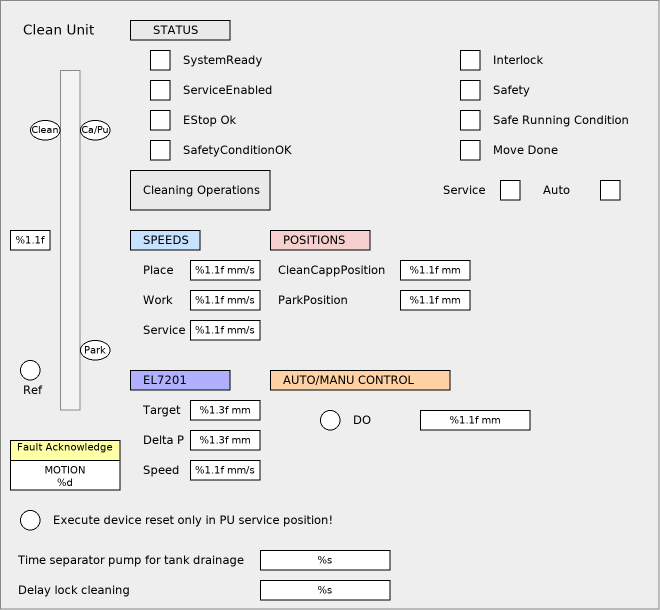
VISUALIZATION _VISU_CLEAN_CU  // 660x610
VAR_IN_OUT
  m_Inst : INT;               (*visu instance*) 
END_VAR
    Rectangle (0,0 660x610)
    Polyline (200,380)
    Rectangle (130,370 100x20)
    Rectangle (270,370 180x20)
    Rectangle (270,230 100x20)
    Rectangle (130,230 70x20)
    Rectangle (280,370 170x20), "AUTO/MANU CONTROL"
    Polyline (440,380)
    Ellipse (20,360 20x20), colour toggle: PRG_MACHINE.fb_CleaningCU[m_Inst].bL_ReferenceSensor
    Rectangle (20,380 30x20), "Ref"
    Scrollbar (60,70 20x340)
        p3598130195: -0.01
        p2245068023: 0.6
        p1057716461: PRG_MACHINE.fb_CleaningCU[m_Inst].fB_Axis.fO_ActualPosition
    Rectangle (10,230 40x20), "%1.1f", text variable: 1000 * PRG_MACHINE.fb_CleaningCU[m_Inst].fB_Axis.fO_ActualPosition
    Rectangle (140,230 70x20), "SPEEDS"
    Polyline (130,240)
    Polyline (340,240)
    Rectangle (280,230 90x20), "POSITIONS"
    Rectangle (190,400 70x20), "%1.3f mm", text variable: 1000 * PRG_MACHINE.fb_CleaningCU[m_Inst].fB_Axis.fI_TargetPosition
    Rectangle (140,400 70x20), "Target"
    Rectangle (140,460 70x20), "Speed"
    Rectangle (190,460 70x20), "%1.1f mm/s", text variable: 1000 * PRG_MACHINE.fb_CleaningCU[m_Inst].fB_Axis.fI_SpeedLimit
    Rectangle (140,370 90x20), "EL7201"
    Rectangle (140,430 70x20), "Delta P"
    Rectangle (190,430 70x20), "%1.3f mm", text variable: 1000 * PRG_MACHINE.fb_CleaningCU[m_Inst].fB_Axis.fL_Delta_P
    Ellipse (30,120 30x20), "Clean", colour toggle: PRG_MACHINE.fb_CleaningCU[m_Inst].pInPosCappingClean
    Ellipse (80,340 30x20), "Park", colour toggle: PRG_MACHINE.fb_CleaningCU[m_Inst].pInPosPark
    Ellipse (80,120 30x20), "Ca/Pu", colour toggle: PRG_MACHINE.fb_CleaningCU[m_Inst].pInPosCappingClean
    Rectangle (20,20 110x20), "Clean Unit"
    Rectangle (10,440 110x50), "Fault Acknowledge", colour toggle: (PRG_MACHINE.fb_CleaningCU[m_Inst].wL_ErrorCode) <> 0
    RoundedRectangle (10,460 110x30), "%d", text variable: PRG_MACHINE.fB_CleaningCU[m_Inst].wL_ErrorCode
        tap PRG_MACHINE.sADS_CleanAxis[iCPr_MAP_Cp_CuAxis[m_Inst]].bI_FaultAck
    RoundedRectangle (10,460 110x20), "MOTION"
    Rectangle (130,170 140x40)
    Rectangle (130,20 100x20)
    Polyline (130,30)
    Polyline (230,30)
    Rectangle (150,20 60x20), "STATUS"
    RoundedRectangle (150,80 20x20), colour toggle: PRG_MACHINE.fb_CleanProcess[m_Inst].bI_UsrService
    RoundedRectangle (150,110 20x20), colour toggle: PRG_MACHINE.bL_IO_EStopOK
    RoundedRectangle (150,140 20x20), colour toggle: PRG_MACHINE.fB_Machine.bI_SafetyOk
    RoundedRectangle (460,140 20x20), colour toggle: NOT PRG_MACHINE.fb_CleaningCU[m_Inst].bL_Busy
    RoundedRectangle (150,50 20x20), colour toggle: PRG_MACHINE.fB_Machine.bI_MachineReady
    Rectangle (180,50 120x20), "SystemReady"
    Rectangle (180,80 120x20), "ServiceEnabled"
    Rectangle (180,110 120x20), "EStop Ok"
    Rectangle (180,140 120x20), "SafetyConditionOK"
    Rectangle (490,140 90x20), "Move Done"
    RoundedRectangle (460,80 20x20), colour toggle: PRG_MACHINE.fb_CleaningCU[m_Inst].bI_SafeToMove
    Rectangle (490,80 120x20), "Safety"
    RoundedRectangle (460,50 20x20), colour toggle: PRG_MACHINE.fb_CleaningCU[m_Inst].bI_SafeToMove
    Rectangle (490,50 120x20), "Interlock"
    Polyline (640,160)
    Rectangle (140,180 140x20), "Cleaning Operations"
    Polyline (270,200)
    RoundedRectangle (460,110 20x20), colour toggle: PRG_MACHINE.fb_CleaningCU[m_Inst].bL_SafeRunningCondition
    Rectangle (490,110 150x20), "Safe Running Condition"
    RoundedRectangle (600,180 20x20), colour toggle: PRG_MACHINE.fb_CleanProcess[m_Inst].bI_UsrAutoMode
    Rectangle (540,180 60x20), "Auto"
    Polyline (340,80)
    RoundedRectangle (500,180 20x20), colour toggle: PRG_MACHINE.fb_CleanProcess[m_Inst].bI_UsrService
    Rectangle (440,180 60x20), "Service"
    Rectangle (420,410 110x20), "%1.1f mm", text variable: PRG_MACHINE.sADS_CleanAxis[iCPr_MAP_Cp_CuAxis[m_Inst]].fI_ManualTargetPos
        OnMouseDown: write the text variable via VisuDialogs.Numpad, min PRG_MACHINE.sADS_CleanAxis[iCPr_MAP_Cp_CuAxis[m_Inst]].sO_AxisPosition.fC_Min, max PRG_MACHINE.sADS_CleanAxis[iCPr_MAP_Cp_CuAxis[m_Inst]].sO_AxisPosition.fC_Max
    Rectangle (350,410 60x20), "DO"
    Ellipse (320,410 20x20), colour toggle: PRG_MACHINE.sADS_CleanAxis[iCPr_MAP_Cp_CuAxis[m_Inst]].bI_ManualMove, input disabled if: NOT PRG_MACHINE.sADS_CleanAxis[iCPr_MAP_Cp_CuAxis[m_Inst]].bO_ManualMoveCanEx
        toggle PRG_MACHINE.sADS_CleanAxis[iCPr_MAP_Cp_CuAxis[m_Inst]].bI_ManualMove
    Rectangle (190,260 70x20), "%1.1f mm/s", text variable: PRG_MACHINE.fb_CleaningCU[m_Inst].sI_SpeedDef.fP_PlaceSpeed
        OnMouseDown: write the text variable via VisuDialogs.Numpad
    Rectangle (190,290 70x20), "%1.1f mm/s", text variable: PRG_MACHINE.fb_CleaningCU[m_Inst].sI_SpeedDef.fP_WorkSpeed
        OnMouseDown: write the text variable via VisuDialogs.Numpad
    Rectangle (190,320 70x20), "%1.1f mm/s", text variable: PRG_MACHINE.fb_CleaningCU[m_Inst].sI_SpeedDef.fP_ServiceSpeed
        OnMouseDown: write the text variable via VisuDialogs.Numpad
    Rectangle (140,260 60x20), "Place"
    Rectangle (140,290 60x20), "Work"
    Rectangle (140,320 60x20), "Service"
    Rectangle (400,260 70x20), "%1.1f mm", text variable: PRG_MACHINE.fb_CleaningCU[m_Inst].fI_PositionCappingClean
        OnMouseDown: write the text variable via VisuDialogs.Numpad
    Rectangle (275,260 125x20), "CleanCappPosition"
    Rectangle (15,550 240x20), "Time separator pump for tank drainage"
    Rectangle (260,550 130x20), "%s", text variable: PRG_MACHINE.tR_TimeSeparatorPump
        OnMouseDown: write the text variable via Default
    Rectangle (400,290 70x20), "%1.1f mm", text variable: PRG_MACHINE.fb_CleaningCU[m_Inst].fI_PositionPark
        OnMouseDown: write the text variable via VisuDialogs.Numpad
    Rectangle (275,290 125x20), "ParkPosition"
    Ellipse (20,510 20x20), colour toggle: PRG_MACHINE.fb_CleaningCU[m_Inst].bIDp_DeviceReset, input disabled if: PRG_MACHINE.fb_CleaningPU[m_Inst].pInPosService
        tap PRG_MACHINE.fb_CleaningCU[m_Inst].bIDp_DeviceReset
    Rectangle (50,510 306x20), "Execute device reset only in PU service position!"
    Rectangle (15,580 240x20), "Delay lock cleaning"
    Rectangle (260,580 130x20), "%s", text variable: PRG_MACHINE.tR_TimeSeparatorLevelCheck
        OnMouseDown: write the text variable via Default
END_VISUALIZATION

(* stored: Version 1.1.0.1, ProductVersion 3.1.4024.9
   Visu _VISU_CLEAN_CU: Id {3097857a-7b28-4218-a333-ba11da124474} *)
